FUNCTION F_GetSystemDateAndTime : DATE_AND_TIME
VAR
	fbGETSYSTEMTIME : GETSYSTEMTIME;
	stFileTime : T_FILETIME;
END_VAR

fbGETSYSTEMTIME(timeLoDW => stFileTime.dwLowDateTime,
				timeHiDW => stFileTime.dwHighDateTime);

F_GetSystemDateAndTime := FILETIME_TO_DT(fileTime := stFileTime);

END_FUNCTION

(* stored: Version 1.1.0.1, ProductVersion 3.1.4024.15
   POU F_GetSystemDateAndTime: Id {108e82b8-77b5-4d7c-9750-43190c973113}, SpecialFunc None *)
